# EPICS autosave request: ADApp/Db/NDEdge_settings.req
$(P)$(R)LowThreshold
$(P)$(R)ThresholdRatio
